PROGRAM PostRemoteData
VAR
	//Query Builder for Document DB
	fbNoSqlQueryBuilder_DocumentDB: FB_NoSQLQueryBuilder_DocumentDB;
	InsertQueryOption: T_QueryOptionDocumentDB_Insert;
	sDocument: STRING (1000);
	sDBName: STRING := 'Datalog';

	//Document json writer
	fbJsonWriter: FB_JsonSaxWriter;
	
	//Query Execution
	fbNoSqlQuery: FB_NoSQLQueryEvt(sNetID:= '', tTimeout:= T#5S);
	myDBID: UDINT := 2;
	TcMessage: I_TcMessage;
END_VAR

IF GlobalData.bLocalGot THEN
	CreateQuery();
	CreateDocument();
	
	IF fbNoSqlQuery.Execute(hDBID:= myDBID, iNoSQLQueryBuilder:= fbNoSqlQueryBuilder_DocumentDB) THEN
		GlobalData.bLocalGot := FALSE;
		GlobalData.bRemotePosted := TRUE;
		IF fbNoSqlQuery.bError THEN
			TcMessage:= fbNoSqlQuery.ipTcResult;
			GlobalData.bLocalGot := TRUE;
			GlobalData.bRemotePosted := FALSE;
		END_IF
	END_IF
END_IF

ACTION CreateDocument:
fbJsonWriter.StartObject();
fbJsonWriter.AddKey('Timestamp');
fbJsonWriter.AddDateTime(GlobalData.aReadStruct.dtTimestamp);
fbJsonWriter.AddKey('Speed');
fbJsonWriter.AddLreal(GlobalData.aReadStruct.rSpeed);
fbJsonWriter.AddKey('Pos');
fbJsonWriter.AddLreal(GlobalData.aReadStruct.rPos);
fbJsonWriter.AddKey('Pulse');
fbJsonWriter.AddBool(GlobalData.aReadStruct.bPulse);
fbJsonWriter.EndObject();
sDocument := fbJsonWriter.GetDocument();
fbJsonWriter.ResetDocument();
END_ACTION

ACTION CreateQuery:
InsertQueryOption.pDocuments := ADR(sDocument);
InsertQueryOption.cbDocuments := SIZEOF(sDocument);

fbNoSqlQueryBuilder_DocumentDB.eQueryType := E_DocumentDbQueryType.InsertOne;
fbNoSqlQueryBuilder_DocumentDB.sCollectionName := sDBName;
fbNoSqlQueryBuilder_DocumentDB.pQueryOptions := ADR(InsertQueryOption);
fbNoSqlQueryBuilder_DocumentDB.cbQueryOptions := SIZEOF(InsertQueryOption);
END_ACTION

END_PROGRAM

(* stored: Version 1.1.0.1, ProductVersion 3.1.4024.4
   POU PostRemoteData: Id {739b46bf-d99f-41e1-a248-f35519a17b2d}, SpecialFunc None
   Action CreateDocument: Id {bb4591cd-873d-4799-aa4b-b85a07d5e57e}
   Action CreateQuery: Id {2655315e-f323-4ad5-bfc9-07379b6667a2} *)
